Fanuc KAREL source: KT00327.KL

PROGRAM KT00327
%NOLOCKGROUP
VAR
  V1: VECTOR
  V2: VECTOR
  OUT: BOOLEAN
BEGIN
  V1.X = 1.0
  V2.Y = 2.0
  V1.X = 1.0
  V2.Y = 2.0
  OUT = V1 <> V2
END KT00327
